PROGRAM StatePatternTest
VAR
	stateManger: StateManager;
	firststate: FirstState;
	secondState: SecondState;
	stateslist: ARRAY[1..2] OF Istate:=[firststate,secondState];
END_VAR


stateManger(statelist := stateslist);
stateManger.RunProcess();

END_PROGRAM

(* stored: Version 1.1.0.1
   POU StatePatternTest: Id {ff2a673d-2cd4-48fe-826b-729eb6dd3bee}, SpecialFunc None *)
